(*			
	RafalOS
	Rafał Osajda		29.10.2025		TC 4024.66
	Metody do konfiguracji MAchine control wywoływane z MachineConfigure z pomocą przekazanego ITF
*)
INTERFACE ITF_MCMachineControlConfigure EXTENDS ITF_Base

METHOD PUBLIC AddHMIManagerFromConfiguration : BOOL
VAR_INPUT
	itfHMIManager			: ITF_BaseGroupElement;
END_VAR
END_METHOD

METHOD PUBLIC AddRequestModeChange : BOOL
VAR_INPUT
	iNumberOfRequest			: INT;
	itfRequest					: ITF_MCRequiredChange;
END_VAR
END_METHOD

METHOD PUBLIC AddRequestStateChange : BOOL
VAR_INPUT
	iNumberOfRequest			: INT;
	itfRequest					: ITF_MCRequiredChange;
END_VAR
END_METHOD

METHOD AddTopElementFromConfiguration : BOOL
VAR_INPUT
	fbTopElement		: ITF_BaseTopElement;
END_VAR
END_METHOD

METHOD PUBLIC SetStartMode
VAR_INPUT
	eStartMode				: E_BaseMachineMode;
END_VAR
END_METHOD

END_INTERFACE

(* stored: Version 1.1.0.1
   Itf ITF_MCMachineControlConfigure: Id {407b3a6e-6e4f-4b87-8313-a53f9cca235d}
   Method AddHMIManagerFromConfiguration: Id {6f7bea06-7a40-0dc1-19c1-ca7e34083a7d}
   Method AddRequestModeChange: Id {b57a036d-1128-0d9e-3e41-4e327c6cc617}
   Method AddRequestStateChange: Id {08c041f6-74b0-0495-1384-b053ecfc16a9}
   Method AddTopElementFromConfiguration: Id {c458ce8f-1021-07a3-1b12-05adfb9f74f9}
   Method SetStartMode: Id {8d345749-18d6-038a-3e39-290be0c31c98} *)
